(* IEC 61131-3 sources: JaccoSigma/tempclass/Class/Crash, 1 file *)

(* ---- Crash.st ---- *)
(*!
<Class
	Name               = "Crash"
	Revision           = "0.0"
	RealtimeTask       = "false"
	CyclicTask         = "false"
	BackgroundTask     = "false"
	Sigmatek           = "false"
	OSInterface        = "false"
	HighPriority       = "false"
	Automatic          = "false"
	UpdateMode         = "Prescan"
	SharedCommandTable = "true"
	Objectsize         = "(370,120)">
	<Channels>
		<Server Name="ServerDint" Visualized="false" Initialize="false" WriteProtected="false" Retentive="false"/>
		<Server Name="ServerUdint" Visualized="false" Initialize="false" WriteProtected="false" Retentive="false"/>
	</Channels>
</Class>
*)
Crash : CLASS
  //Servers:
	ServerDint 	: SvrChCmd_DINT;
	ServerUdint 	: SvrCh_UDINT;
  //Clients:
  //Variables:
		counter 	: DINT;
		idx2 	: DINT;
		idx 	: UDINT;
  //Functions:

	FUNCTION VIRTUAL GLOBAL ServerDint::Write
		VAR_INPUT
			input (EAX) 	: DINT;
		END_VAR
		VAR_OUTPUT
			result (EAX) 	: DINT;
		END_VAR;

	FUNCTION VIRTUAL GLOBAL ServerUdint::Write
		VAR_INPUT
			input (EAX) 	: UDINT;
		END_VAR
		VAR_OUTPUT
			result (EAX) 	: UDINT;
		END_VAR;
  //Tables:
	FUNCTION @STD
		VAR_OUTPUT
			ret_code	: CONFSTATES;
		END_VAR;
	FUNCTION GLOBAL TAB @CT_;
END_CLASS;

FUNCTION VIRTUAL GLOBAL Crash::ServerDint::Write
	VAR_INPUT
		input (EAX) 	: DINT;
	END_VAR
	VAR_OUTPUT
		result (EAX) 	: DINT;
	END_VAR

	ServerDint := input;
  counter := 0;

  FOR Idx2:=10 TO 0 BY -1 DO
    if IDX2>10 then
      ServerDint:=idx2;
    end_if;
  counter += 1;
  END_FOR;

	result := ServerDint;

END_FUNCTION

FUNCTION VIRTUAL GLOBAL Crash::ServerUdint::Write
	VAR_INPUT
		input (EAX) 	: UDINT;
	END_VAR
	VAR_OUTPUT
		result (EAX) 	: UDINT;
	END_VAR

	ServerUdint := input;

  counter := 0;

  FOR Idx:=10 TO 0 BY -1 DO
    if IDX>10 then
      ServerUdint:=idx;
    end_if;
  counter += 1;
  END_FOR;

	result := ServerUdint;

END_FUNCTION
